// TIA Portal V19 export
ORGANIZATION_BLOCK "TOD_INT1"   // OB10, STL, TimeOfDay
TITLE = "Time of Day Interrupt"
{ S7_Optimized_Access := 'TRUE' }
VERSION : 0.0
// Comment
// stored: AutoNumber false
   VAR_INPUT
      CaughtUp : Bool;   // OB call is caught up because time was set forward
      SecondTime : Bool;   // OB call is started a second time because time was set backward
   END_VAR
BEGIN
END_ORGANIZATION_BLOCK
